// TIA Portal V16 export
// export: Created 2021-03-04T22:04:03.336434Z, ExportSetting WithDefaults, DisplayName Totally Integrated Automation Portal, DisplayVersion V16, DisplayName TIA Portal Version Control Interface, DisplayVersion V16, DisplayName TIA Portal Openness, DisplayVersion V16, DisplayName SINAMICS Startdrive Advanced, DisplayVersion V16, DisplayName SINAMICS Startdrive G130, G150, S120, S150, SINAMICS MV, S210, DisplayVersion V16, DisplayName SINAMICS Startdrive G110M, G120, G120C, G120D, G120P, DisplayVersion V16, DisplayName STEP 7 Professional, DisplayVersion V16, DisplayName STEP 7 Safety, DisplayVersion V16, DisplayName WinCC Professional, DisplayVersion V16
FUNCTION "fcSetHMIStatusSimulation" : Void   // FC333, LAD
TITLE = Sets HMI Status
{ S7_Optimized_Access := 'TRUE' }
VERSION : 0.1
// Wrapper function for setting the HMI status of a device
// 
// In order of priority:
// 1. E-stop
// 2. Error
// 3. Forward/Work Position
// 4. Reverse/Home Position
// 5. Forward/Work On
// 6. Reverse/Home On
// 7. None
// stored: AutoNumber true, IsIECCheckEnabled false, SetENOAutomatically false, UDAEnableTagReadback false
   VAR_INPUT
      bInEstop : Bool;
      bInError : Bool;
      bInForwardWork : Bool;
      bInReverseHome : Bool;
      bInOnForwardWork : Bool;
      bInOnReverseHome : Bool;
      bInSimulate : Bool;
   END_VAR
   VAR_OUTPUT
      iOutStatus : Int;
   END_VAR
BEGIN

REGION Network 1: Set Reverse/Home On
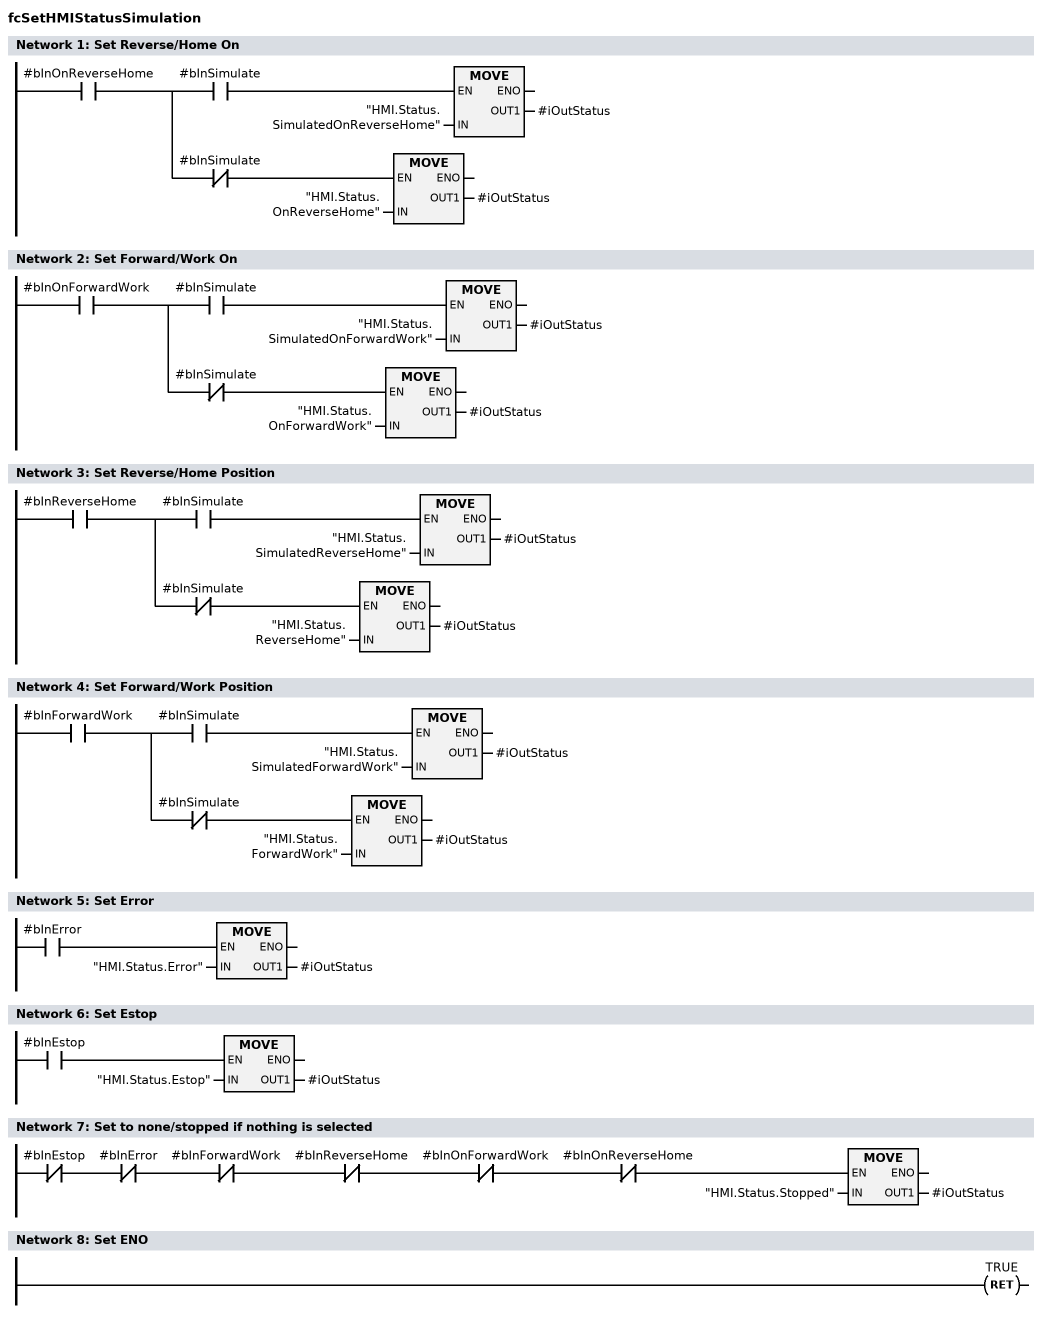
   RUNG wire#powerrail
      Contact( #bInOnReverseHome )
      wire#w1
      Contact( #bInSimulate )
      Move(in := "HMI.Status.SimulatedOnReverseHome", out1 => #iOutStatus)
   END_RUNG
   RUNG wire#w1
      I_Contact( #bInSimulate )
      Move(in := "HMI.Status.OnReverseHome", out1 => #iOutStatus)
   END_RUNG
   // the same network as SCL:
   IF #bInOnReverseHome AND #bInSimulate THEN #iOutStatus := "HMI.Status.SimulatedOnReverseHome"; END_IF;
   IF #bInOnReverseHome AND NOT #bInSimulate THEN #iOutStatus := "HMI.Status.OnReverseHome"; END_IF;
END_REGION

REGION Network 2: Set Forward/Work On
   RUNG wire#powerrail
      Contact( #bInOnForwardWork )
      wire#w1
      Contact( #bInSimulate )
      Move(in := "HMI.Status.SimulatedOnForwardWork", out1 => #iOutStatus)
   END_RUNG
   RUNG wire#w1
      I_Contact( #bInSimulate )
      Move(in := "HMI.Status.OnForwardWork", out1 => #iOutStatus)
   END_RUNG
   // the same network as SCL:
   IF #bInOnForwardWork AND #bInSimulate THEN #iOutStatus := "HMI.Status.SimulatedOnForwardWork"; END_IF;
   IF #bInOnForwardWork AND NOT #bInSimulate THEN #iOutStatus := "HMI.Status.OnForwardWork"; END_IF;
END_REGION

REGION Network 3: Set Reverse/Home Position
   RUNG wire#powerrail
      Contact( #bInReverseHome )
      wire#w1
      Contact( #bInSimulate )
      Move(in := "HMI.Status.SimulatedReverseHome", out1 => #iOutStatus)
   END_RUNG
   RUNG wire#w1
      I_Contact( #bInSimulate )
      Move(in := "HMI.Status.ReverseHome", out1 => #iOutStatus)
   END_RUNG
   // the same network as SCL:
   IF #bInReverseHome AND #bInSimulate THEN #iOutStatus := "HMI.Status.SimulatedReverseHome"; END_IF;
   IF #bInReverseHome AND NOT #bInSimulate THEN #iOutStatus := "HMI.Status.ReverseHome"; END_IF;
END_REGION

REGION Network 4: Set Forward/Work Position
   RUNG wire#powerrail
      Contact( #bInForwardWork )
      wire#w1
      Contact( #bInSimulate )
      Move(in := "HMI.Status.SimulatedForwardWork", out1 => #iOutStatus)
   END_RUNG
   RUNG wire#w1
      I_Contact( #bInSimulate )
      Move(in := "HMI.Status.ForwardWork", out1 => #iOutStatus)
   END_RUNG
   // the same network as SCL:
   IF #bInForwardWork AND #bInSimulate THEN #iOutStatus := "HMI.Status.SimulatedForwardWork"; END_IF;
   IF #bInForwardWork AND NOT #bInSimulate THEN #iOutStatus := "HMI.Status.ForwardWork"; END_IF;
END_REGION

REGION Network 5: Set Error
   RUNG wire#powerrail
      Contact( #bInError )
      Move(in := "HMI.Status.Error", out1 => #iOutStatus)
   END_RUNG
   // the same network as SCL:
   IF #bInError THEN #iOutStatus := "HMI.Status.Error"; END_IF;
END_REGION

REGION Network 6: Set Estop
   RUNG wire#powerrail
      Contact( #bInEstop )
      Move(in := "HMI.Status.Estop", out1 => #iOutStatus)
   END_RUNG
   // the same network as SCL:
   IF #bInEstop THEN #iOutStatus := "HMI.Status.Estop"; END_IF;
END_REGION

REGION Network 7: Set to none/stopped if nothing is selected
   RUNG wire#powerrail
      I_Contact( #bInEstop )
      I_Contact( #bInError )
      I_Contact( #bInForwardWork )
      I_Contact( #bInReverseHome )
      I_Contact( #bInOnForwardWork )
      I_Contact( #bInOnReverseHome )
      Move(in := "HMI.Status.Stopped", out1 => #iOutStatus)
   END_RUNG
   // the same network as SCL:
   IF NOT #bInEstop AND NOT #bInError AND NOT #bInForwardWork AND NOT #bInReverseHome AND NOT #bInOnForwardWork AND NOT #bInOnReverseHome THEN
       #iOutStatus := "HMI.Status.Stopped";
   END_IF;
END_REGION

REGION Network 8: Set ENO
   RUNG wire#powerrail
      ReturnCoil( TRUE )
   END_RUNG
   // the same network as SCL:
   ENO := TRUE;
   RETURN;
END_REGION
END_FUNCTION
